// Mitsubishi GX Works2 project: PLCtoPCexample   PLC: Q04UDH

PROGRAM MAIN
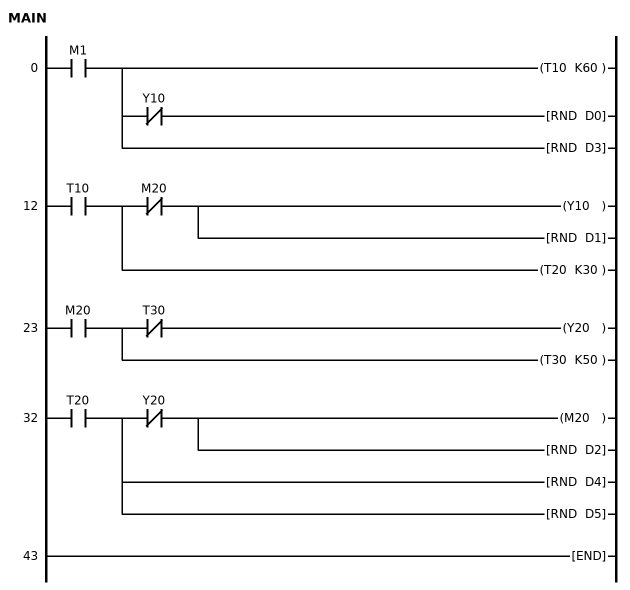
0     LD      M1
      OUT     T10 K60
      MPS
      ANI     Y10
      RND     D0
      MPP
      RND     D3
12    LD      T10
      MPS
      ANI     M20
      OUT     Y10
      RND     D1
      MPP
      OUT     T20 K30
23    LD      M20
      MPS
      ANI     T30
      OUT     Y20
      MPP
      OUT     T30 K50
32    LD      T20
      MPS
      ANI     Y20
      OUT     M20
      RND     D2
      MPP
      RND     D4
      RND     D5
43    END
END_PROGRAM
